// Basic empty interface, no inheritance, no methods no properties.
INTERFACE I_Empty

END_INTERFACE

(* stored: Version 1.1.0.1, ProductVersion 3.1.4024.15
   Itf I_Empty: Id {1b7d3ab1-e50f-48d0-87d7-12bc0240a7e1} *)
